(* CoDeSys 2.3 export: F_READ_SENSOR_POS.EXP *)

(* POU FUN/PARAMETERS/F_READ_SENSOR_POS, ST *)
FUNCTION F_READ_SENSOR_POS : BOOL
VAR_INPUT
END_VAR
VAR_IN_OUT
	stSensor : ST_SENSOR_POS;
	fbIdList : FB_IDLIST;
END_VAR
VAR
END_VAR
stSensor.Cal_K   := F_IDLIST_GETREAL( CONCAT(stSensor.Name, '_K'   ), fbIdList );
stSensor.Cal_Off := F_IDLIST_GETREAL( CONCAT(stSensor.Name, '_Off' ), fbIdList );
END_FUNCTION
